{attribute 'qualified_only'}
VAR_GLOBAL
	myTimer		:FB_Timer;
END_VAR

(* stored: Version 1.1.0.1, ProductVersion 3.1.4022.16
   GVL GVL_General: Id {76c8226e-a857-4248-bb6f-45b7b244b07e} *)
